ADAPTER ASR (* unidirectional Adapter Interface for 2 Events *)
  (* Standard: 61499-1 *)
  (* Version 1.0, 2025-05-27, franz *)
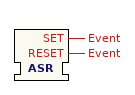
  EVENT_OUTPUT
    SET; (* Set / Switch on *)
    RESET; (* Reset / Switch off *)
  END_EVENT
END_ADAPTER
